PROGRAM P_Demo_OnAlarmConfirmed
VAR
    fbListener : FB_ListenerBase2; // listener 实例（实际工程使用子类）
END_VAR

// =============================================================================
// 场景：覆盖（OVERRIDE）OnAlarmConfirmed 回调记录事件元数据到内部计数器
// 价值：事件驱动接收的最小实现
// 验证：本回调由 EventLogger 在事件发生时自动调用——不能在主程序里手动调用做演示。实际工程：继承 FB_ListenerBase2 后 OVERRIDE 本方法，再让事件触发
// 验证步骤：
//   1. 右键 PLC 项目下 POUs 文件夹 → Add → Existing Item → 选本 .TcPOU 文件
//   2. 引用 Tc3_EventLogger（System → References → Add library）
//   3. 编译 → 登录 → 运行；按 verify 注释里给出的在线写值操作
// =============================================================================

// 本方法是 EventLogger 的事件回调，应该在 FB_ListenerBase2 的子类里 OVERRIDE。
// 这里仅展示在主程序里启动 listener 的代码骨架；具体 OnAlarmConfirmed 重写见同名 METHOD。
// 示例（仅说明）：在子类 FB 里写——
//   METHOD OnAlarmConfirmed : HRESULT
//   VAR_INPUT
//       fbEvent : REFERENCE TO FB_TcEvent;
//   END_VAR
//   nEventCount := nEventCount + 1;
//   OnAlarmConfirmed := S_OK;
//
// 主程序示意：
fbListener.Execute();

END_PROGRAM

(* stored: Version 1.1.0.1, ProductVersion 3.1.4024.5
   POU P_Demo_OnAlarmConfirmed: Id {84f8cd47-9c83-5030-88c8-bded09276d2c}, SpecialFunc None *)
